// TIA Portal V15.1 export
// export: Created 2022-03-15T12:28:27.7152417Z, ExportSetting WithDefaults, WithReadOnly, DisplayName Totally Integrated Automation Portal, DisplayVersion V15.1 Update 3, DisplayName TIA Portal Openness, DisplayVersion V15.1, DisplayName TIA Portal Teamcenter Gateway, DisplayVersion V15.1, DisplayName SINAMICS Startdrive Advanced, DisplayVersion V15.1, DisplayName G130, G150, S120, S150, SINAMICS MV, S210, DisplayVersion V15.1, DisplayName G110M, G120, G120C, G120D, G120P, DisplayVersion V15.1, DisplayName STEP 7 Professional, DisplayVersion V15.1 Update 3, DisplayName STEP 7 Safety, DisplayVersion V15.1, DisplayName WinCC Advanced, DisplayVersion V15.1 Update 3
FUNCTION "Baustein_2" : Void   // FC2, LAD
{ S7_Optimized_Access := 'TRUE' }
VERSION : 0.1
// stored: AutoNumber true, CodeModifiedDate 2022-03-08T11:13:52.6871257Z, CompileDate 2022-03-08T11:13:55.7033463Z, CreationDate 2022-03-08T11:10:33.1505035Z, HandleErrorsWithinBlock false, InterfaceModifiedDate 2022-03-08T11:10:33.1505035Z, IsConsistent true, IsIECCheckEnabled false, IsKnowHowProtected false, IsWriteProtected false, LibraryConformanceStatus Fehler: Der Baustein enthält Aufrufe von Einzelinstanzen. Warnung: Der Baustein enthält direkte Zugriffe auf Eingänge, Ausgänge, Merker, indirekte Zugriffe auf Register oder indirekte Zugriffe auf externe, zum Übersetzungszeitpunkt unbekannte Speicherbereiche., ModifiedDate 2022-03-08T11:13:52.6871257Z, ParameterModified 2022-03-08T11:10:33.1505035Z, PLCSimAdvancedSupport false, SetENOAutomatically False, StructureModified 2022-03-08T11:10:33.1505035Z, UDAEnableTagReadback false
BEGIN

REGION Network 1
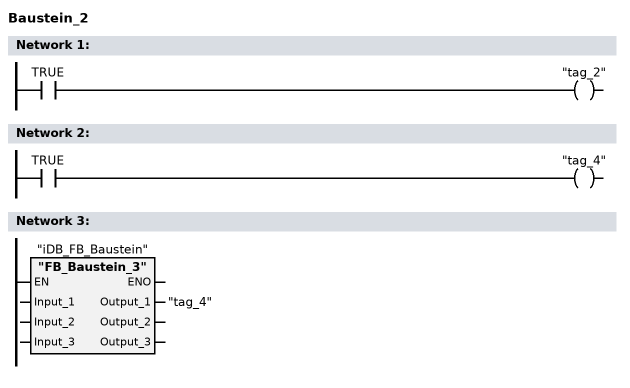
   RUNG wire#powerrail
      Contact( TRUE )
      Coil( "tag_2" )
   END_RUNG
   // the same network as SCL:
   "tag_2" := TRUE;
END_REGION

REGION Network 2
   RUNG wire#powerrail
      Contact( TRUE )
      Coil( "tag_4" )
   END_RUNG
   // the same network as SCL:
   "tag_4" := TRUE;
END_REGION

REGION Network 3
   RUNG wire#powerrail
      "iDB_FB_Baustein"(Input_1 :=, Input_2 :=, Input_3 :=, Output_1 => "tag_4", Output_2 =>, Output_3 =>)
   END_RUNG
   // the same network as SCL:
   "iDB_FB_Baustein"(Output_1 => "tag_4");   // "FB_Baustein_3"
END_REGION
END_FUNCTION
